(* IEC 61131-3 sources: AXOpen/src/template.axolibrary/app/src/Sandbox, 1 file *)

(* ---- SandboxContext.st ---- *)
USING AXOpen.Core;
NAMESPACE Template.Axolibrary
    {S7.extern=ReadWrite}
    CLASS SandboxContext EXTENDS AXOpen.Core.AxoContext
        VAR PUBLIC
            _manualControl : BOOL;
            _testCyclinder : Template.Axolibrary.TemplateComponent;
            _homeSensor : BOOL;
            _workSensor : BOOL;
            _moveHomeSignal : BOOL;
            _moveWorkSignal : BOOL;
            _rootObject : AxoObject;
        END_VAR

        METHOD PROTECTED OVERRIDE Main
            THIS.InitializeRootObject(_rootObject);
            _testCyclinder.Run(_rootObject,
                                WORD#64,
                                REF(_homeSensor),
                                REF(_workSensor),
                                REF(_moveHomeSignal),
                                REF(_moveWorkSignal));

            IF(_manualControl) THEN
                _testCyclinder.ActivateManualControl();
            END_IF;
        END_METHOD
    END_CLASS
END_NAMESPACE
